PROGRAM MAIN
VAR
END_VAR

END_PROGRAM

(* stored: Version 1.1.0.1
   POU MAIN: Id {56f4075e-4895-4e88-bf82-4d98b9642bb1} *)
